Fanuc KAREL source: PIPE_CONFIG.kl

PROGRAM T
%NOLOCKGROUP
VAR
 v0 : STRING[40]
 v1 : BOOLEAN
 v2 : INTEGER
 v3 : INTEGER
 v4 : STRING[40]
 v5 : INTEGER
 v6 : INTEGER
BEGIN
 PIPE_CONFIG(v0, v1, v2, v3, v4, v5, v6)
END T
